FUNCTION_BLOCK cPressControl (* Composite Function Block Type *)
  (* Standard: 61499-2 *)
  (* Version 0.0, 26/03/2026, template *)
  PACKAGE Hidryco.HidrycoLib;
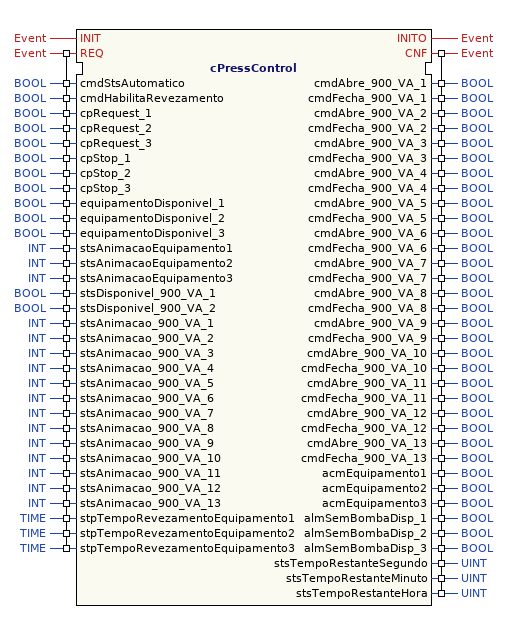
  EVENT_INPUT
    INIT; (* Initialization Request *)
    REQ WITH cmdStsAutomatico, cmdHabilitaRevezamento, cpRequest_1, cpRequest_2, cpRequest_3, cpStop_1, cpStop_2, cpStop_3, equipamentoDisponivel_1, equipamentoDisponivel_2, equipamentoDisponivel_3, stsAnimacaoEquipamento1, stsAnimacaoEquipamento2, stsAnimacaoEquipamento3, stsDisponivel_900_VA_1, stsDisponivel_900_VA_2, stsAnimacao_900_VA_1, stsAnimacao_900_VA_2, stsAnimacao_900_VA_3, stsAnimacao_900_VA_4, stsAnimacao_900_VA_5, stsAnimacao_900_VA_6, stsAnimacao_900_VA_7, stsAnimacao_900_VA_8, stsAnimacao_900_VA_9, stsAnimacao_900_VA_10, stsAnimacao_900_VA_11, stsAnimacao_900_VA_12, stsAnimacao_900_VA_13, stpTempoRevezamentoEquipamento1, stpTempoRevezamentoEquipamento2, stpTempoRevezamentoEquipamento3; (* Normal Execution Request *)
  END_EVENT
  EVENT_OUTPUT
    INITO; (* Initialization Confirm *)
    CNF WITH cmdAbre_900_VA_1, cmdFecha_900_VA_1, cmdAbre_900_VA_2, cmdFecha_900_VA_2, cmdAbre_900_VA_3, cmdFecha_900_VA_3, cmdAbre_900_VA_4, cmdFecha_900_VA_4, cmdAbre_900_VA_5, cmdFecha_900_VA_5, cmdAbre_900_VA_6, cmdFecha_900_VA_6, cmdAbre_900_VA_7, cmdFecha_900_VA_7, cmdAbre_900_VA_8, cmdFecha_900_VA_8, cmdAbre_900_VA_9, cmdFecha_900_VA_9, cmdAbre_900_VA_10, cmdFecha_900_VA_10, cmdAbre_900_VA_11, cmdFecha_900_VA_11, cmdAbre_900_VA_12, cmdFecha_900_VA_12, cmdAbre_900_VA_13, cmdFecha_900_VA_13, acmEquipamento1, acmEquipamento2, acmEquipamento3, almSemBombaDisp_1, almSemBombaDisp_2, almSemBombaDisp_3, stsTempoRestanteSegundo, stsTempoRestanteMinuto, stsTempoRestanteHora; (* Execution Confirmation *)
  END_EVENT
  VAR_INPUT
    cmdStsAutomatico : BOOL;
    cmdHabilitaRevezamento : BOOL;
    cpRequest_1 : BOOL;
    cpRequest_2 : BOOL;
    cpRequest_3 : BOOL;
    cpStop_1 : BOOL;
    cpStop_2 : BOOL;
    cpStop_3 : BOOL;
    equipamentoDisponivel_1 : BOOL;
    equipamentoDisponivel_2 : BOOL;
    equipamentoDisponivel_3 : BOOL;
    stsAnimacaoEquipamento1 : INT;
    stsAnimacaoEquipamento2 : INT;
    stsAnimacaoEquipamento3 : INT;
    stsDisponivel_900_VA_1 : BOOL;
    stsDisponivel_900_VA_2 : BOOL;
    stsAnimacao_900_VA_1 : INT;
    stsAnimacao_900_VA_2 : INT;
    stsAnimacao_900_VA_3 : INT;
    stsAnimacao_900_VA_4 : INT;
    stsAnimacao_900_VA_5 : INT;
    stsAnimacao_900_VA_6 : INT;
    stsAnimacao_900_VA_7 : INT;
    stsAnimacao_900_VA_8 : INT;
    stsAnimacao_900_VA_9 : INT;
    stsAnimacao_900_VA_10 : INT;
    stsAnimacao_900_VA_11 : INT;
    stsAnimacao_900_VA_12 : INT;
    stsAnimacao_900_VA_13 : INT;
    stpTempoRevezamentoEquipamento1 : TIME;
    stpTempoRevezamentoEquipamento2 : TIME;
    stpTempoRevezamentoEquipamento3 : TIME;
  END_VAR
  VAR_OUTPUT
    cmdAbre_900_VA_1 : BOOL;
    cmdFecha_900_VA_1 : BOOL;
    cmdAbre_900_VA_2 : BOOL;
    cmdFecha_900_VA_2 : BOOL;
    cmdAbre_900_VA_3 : BOOL;
    cmdFecha_900_VA_3 : BOOL;
    cmdAbre_900_VA_4 : BOOL;
    cmdFecha_900_VA_4 : BOOL;
    cmdAbre_900_VA_5 : BOOL;
    cmdFecha_900_VA_5 : BOOL;
    cmdAbre_900_VA_6 : BOOL;
    cmdFecha_900_VA_6 : BOOL;
    cmdAbre_900_VA_7 : BOOL;
    cmdFecha_900_VA_7 : BOOL;
    cmdAbre_900_VA_8 : BOOL;
    cmdFecha_900_VA_8 : BOOL;
    cmdAbre_900_VA_9 : BOOL;
    cmdFecha_900_VA_9 : BOOL;
    cmdAbre_900_VA_10 : BOOL;
    cmdFecha_900_VA_10 : BOOL;
    cmdAbre_900_VA_11 : BOOL;
    cmdFecha_900_VA_11 : BOOL;
    cmdAbre_900_VA_12 : BOOL;
    cmdFecha_900_VA_12 : BOOL;
    cmdAbre_900_VA_13 : BOOL;
    cmdFecha_900_VA_13 : BOOL;
    acmEquipamento1 : BOOL;
    acmEquipamento2 : BOOL;
    acmEquipamento3 : BOOL;
    almSemBombaDisp_1 : BOOL;
    almSemBombaDisp_2 : BOOL;
    almSemBombaDisp_3 : BOOL;
    stsTempoRestanteSegundo : UINT;
    stsTempoRestanteMinuto : UINT;
    stsTempoRestanteHora : UINT;
  END_VAR
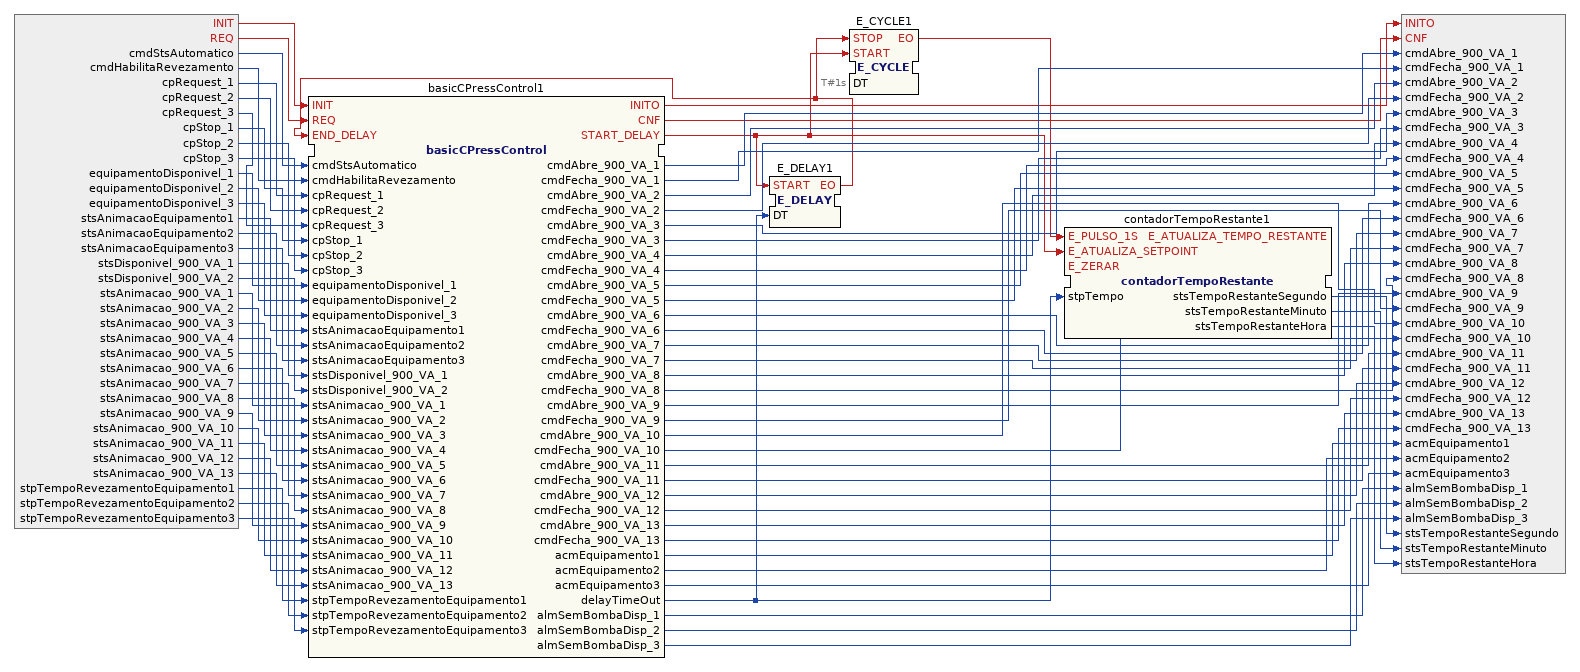
  FBS
    basicCPressControl1 : basicCPressControl;
    E_DELAY1 : E_DELAY;
    E_CYCLE1 : E_CYCLE(DT := T#1s);
    contadorTempoRestante1 : contadorTempoRestante;
  END_FBS
  EVENT_CONNECTIONS
    basicCPressControl1.INITO TO INITO;
    basicCPressControl1.CNF TO CNF;
    INIT TO basicCPressControl1.INIT;
    REQ TO basicCPressControl1.REQ;
    E_DELAY1.EO TO E_CYCLE1.STOP;
    basicCPressControl1.START_DELAY TO E_DELAY1.START;
    basicCPressControl1.START_DELAY TO E_CYCLE1.START;
    E_CYCLE1.EO TO contadorTempoRestante1.E_PULSO_1S;
    basicCPressControl1.START_DELAY TO contadorTempoRestante1.E_ATUALIZA_SETPOINT;
    E_DELAY1.EO TO basicCPressControl1.END_DELAY;
  END_CONNECTIONS
  DATA_CONNECTIONS
    basicCPressControl1.delayTimeOut TO E_DELAY1.DT;
    basicCPressControl1.delayTimeOut TO contadorTempoRestante1.stpTempo;
    cmdStsAutomatico TO basicCPressControl1.cmdStsAutomatico;
    cmdHabilitaRevezamento TO basicCPressControl1.cmdHabilitaRevezamento;
    cpRequest_1 TO basicCPressControl1.cpRequest_1;
    cpRequest_2 TO basicCPressControl1.cpRequest_2;
    stpTempoRevezamentoEquipamento3 TO basicCPressControl1.stpTempoRevezamentoEquipamento3;
    stpTempoRevezamentoEquipamento2 TO basicCPressControl1.stpTempoRevezamentoEquipamento2;
    stpTempoRevezamentoEquipamento1 TO basicCPressControl1.stpTempoRevezamentoEquipamento1;
    stsAnimacao_900_VA_13 TO basicCPressControl1.stsAnimacao_900_VA_13;
    stsAnimacao_900_VA_12 TO basicCPressControl1.stsAnimacao_900_VA_12;
    stsAnimacao_900_VA_11 TO basicCPressControl1.stsAnimacao_900_VA_11;
    stsAnimacao_900_VA_10 TO basicCPressControl1.stsAnimacao_900_VA_10;
    stsAnimacao_900_VA_9 TO basicCPressControl1.stsAnimacao_900_VA_9;
    stsAnimacao_900_VA_8 TO basicCPressControl1.stsAnimacao_900_VA_8;
    stsAnimacao_900_VA_7 TO basicCPressControl1.stsAnimacao_900_VA_7;
    stsAnimacao_900_VA_6 TO basicCPressControl1.stsAnimacao_900_VA_6;
    stsAnimacao_900_VA_5 TO basicCPressControl1.stsAnimacao_900_VA_5;
    stsAnimacao_900_VA_4 TO basicCPressControl1.stsAnimacao_900_VA_4;
    stsAnimacao_900_VA_3 TO basicCPressControl1.stsAnimacao_900_VA_3;
    stsAnimacao_900_VA_2 TO basicCPressControl1.stsAnimacao_900_VA_2;
    stsAnimacao_900_VA_1 TO basicCPressControl1.stsAnimacao_900_VA_1;
    stsDisponivel_900_VA_2 TO basicCPressControl1.stsDisponivel_900_VA_2;
    stsDisponivel_900_VA_1 TO basicCPressControl1.stsDisponivel_900_VA_1;
    stsAnimacaoEquipamento3 TO basicCPressControl1.stsAnimacaoEquipamento3;
    stsAnimacaoEquipamento2 TO basicCPressControl1.stsAnimacaoEquipamento2;
    stsAnimacaoEquipamento1 TO basicCPressControl1.stsAnimacaoEquipamento1;
    equipamentoDisponivel_3 TO basicCPressControl1.equipamentoDisponivel_3;
    equipamentoDisponivel_2 TO basicCPressControl1.equipamentoDisponivel_2;
    equipamentoDisponivel_1 TO basicCPressControl1.equipamentoDisponivel_1;
    cpStop_3 TO basicCPressControl1.cpStop_3;
    cpStop_2 TO basicCPressControl1.cpStop_2;
    cpStop_1 TO basicCPressControl1.cpStop_1;
    cpRequest_3 TO basicCPressControl1.cpRequest_3;
    basicCPressControl1.cmdAbre_900_VA_1 TO cmdAbre_900_VA_1;
    basicCPressControl1.cmdFecha_900_VA_1 TO cmdFecha_900_VA_1;
    basicCPressControl1.cmdAbre_900_VA_2 TO cmdAbre_900_VA_2;
    basicCPressControl1.cmdFecha_900_VA_2 TO cmdFecha_900_VA_2;
    basicCPressControl1.cmdAbre_900_VA_3 TO cmdAbre_900_VA_3;
    basicCPressControl1.cmdFecha_900_VA_3 TO cmdFecha_900_VA_3;
    basicCPressControl1.cmdAbre_900_VA_4 TO cmdAbre_900_VA_4;
    basicCPressControl1.cmdFecha_900_VA_4 TO cmdFecha_900_VA_4;
    basicCPressControl1.cmdAbre_900_VA_5 TO cmdAbre_900_VA_5;
    basicCPressControl1.cmdFecha_900_VA_5 TO cmdFecha_900_VA_5;
    basicCPressControl1.cmdAbre_900_VA_6 TO cmdAbre_900_VA_6;
    basicCPressControl1.cmdFecha_900_VA_6 TO cmdFecha_900_VA_6;
    basicCPressControl1.cmdAbre_900_VA_7 TO cmdAbre_900_VA_7;
    basicCPressControl1.cmdFecha_900_VA_7 TO cmdFecha_900_VA_7;
    basicCPressControl1.cmdAbre_900_VA_8 TO cmdAbre_900_VA_8;
    basicCPressControl1.cmdFecha_900_VA_8 TO cmdFecha_900_VA_8;
    basicCPressControl1.cmdAbre_900_VA_9 TO cmdAbre_900_VA_9;
    basicCPressControl1.cmdFecha_900_VA_9 TO cmdFecha_900_VA_9;
    basicCPressControl1.cmdAbre_900_VA_10 TO cmdAbre_900_VA_10;
    basicCPressControl1.cmdFecha_900_VA_10 TO cmdFecha_900_VA_10;
    basicCPressControl1.cmdAbre_900_VA_11 TO cmdAbre_900_VA_11;
    basicCPressControl1.cmdFecha_900_VA_11 TO cmdFecha_900_VA_11;
    basicCPressControl1.cmdAbre_900_VA_12 TO cmdAbre_900_VA_12;
    basicCPressControl1.cmdFecha_900_VA_12 TO cmdFecha_900_VA_12;
    basicCPressControl1.cmdAbre_900_VA_13 TO cmdAbre_900_VA_13;
    basicCPressControl1.cmdFecha_900_VA_13 TO cmdFecha_900_VA_13;
    basicCPressControl1.acmEquipamento1 TO acmEquipamento1;
    basicCPressControl1.acmEquipamento2 TO acmEquipamento2;
    basicCPressControl1.acmEquipamento3 TO acmEquipamento3;
    basicCPressControl1.almSemBombaDisp_1 TO almSemBombaDisp_1;
    basicCPressControl1.almSemBombaDisp_2 TO almSemBombaDisp_2;
    basicCPressControl1.almSemBombaDisp_3 TO almSemBombaDisp_3;
    contadorTempoRestante1.stsTempoRestanteSegundo TO stsTempoRestanteSegundo;
    contadorTempoRestante1.stsTempoRestanteMinuto TO stsTempoRestanteMinuto;
    contadorTempoRestante1.stsTempoRestanteHora TO stsTempoRestanteHora;
  END_CONNECTIONS
END_FUNCTION_BLOCK
